// TIA Portal V20 export
TYPE "UDT_Flowmeter_Steuern"
   STRUCT
      offset : Real;
      sim : Real;
      Res1 : Int;
      Res2 : Int;
      Sim_FG : Bool;   // Freigabe simulation Value
      Bit0_1 : Bool;
      Bit0_2 : Bool;
      Bit0_3 : Bool;
      Bit0_4 : Bool;
      Bit0_5 : Bool;
      Bit0_6 : Bool;
      Bit0_7 : Bool;
      Bit1_0 : Bool;
      Bit1_1 : Bool;
      Bit1_2 : Bool;
      Bit1_3 : Bool;
      Bit1_4 : Bool;
      Bit1_5 : Bool;
      Bit1_6 : Bool;
      Bit1_7 : Bool;
   END_STRUCT;
END_TYPE
